FUNCTION_BLOCK FB_SimulatedIn_DG IMPLEMENTS ITF_Regelschuif_In_DG

VAR
	internalState : sint;
END_VAR

{warning 'Add method implementation '}
METHOD get : SINT
get := internalState;
END_METHOD

END_FUNCTION_BLOCK

(* stored: Version 1.1.0.1, ProductVersion 3.1.4026.8
   POU FB_SimulatedIn_DG: Id {1937c0a8-07f6-4296-bab0-27257a63d4d8}, SpecialFunc None
   Method get: Id {74e86409-c405-4759-a251-5fa15e22afc3} *)
